// TIA Portal V16 export
// export: Created 2022-11-17T15:49:44.8072382Z, ExportSetting WithDefaults, DisplayName Totally Integrated Automation Portal, DisplayVersion V16 Update 6, DisplayName TIA Portal Version Control Interface, DisplayVersion V16 Update 2, DisplayName TIA Portal Openness, DisplayVersion V16 Update 6, DisplayName SINAMICS Startdrive Advanced, DisplayVersion V16 Update 5, DisplayName SINAMICS Startdrive G130, G150, S120, S150, SINAMICS MV, S210, DisplayVersion V16 Update 5, DisplayName SINAMICS Startdrive G110M, G120, G120C, G120D, G120P, G115D, DisplayVersion V16 Update 5, DisplayName STEP 7 Professional, DisplayVersion V16 Update 6, DisplayName STEP 7 Safety, DisplayVersion V16, DisplayName WinCC Advanced, DisplayVersion V16 Update 6
DATA_BLOCK "DB242_Program8"   // DB242
{ S7_Optimized_Access := 'FALSE' }
AUTHOR : Robopac
VERSION : 0.0
// stored: AutoNumber false, IsOnlyStoredInLoadMemory false, IsWriteProtectedInAS false
   VAR RETAIN
      Program8 { S7_SetPoint := 'True'} : "DatiProgramma";
   END_VAR
BEGIN
   Program8.Wrapping := TRUE;
   Program8.TopLenght := 500;
   Program8.TopRelease := 0;
   Program8.TopDown := 0;
   Program8.Top := 4;
   Program8.PressurePTime := 0;
   Program8.LifterTime := 0;
   Program8.RevOverContrast := 1;
   Program8.RopeEndCycle := 16#02;
   Program8.Spare4 := 16#01;
   Program8.RopeTime := 1500;
   Program8.RevOverClamp := 1;
   Program8.FilmForceFinalRev := 10;
   Program8.FilmPrestretchFinalRev := 100;
   Program8.ArmSpeed := 100;
   Program8.CarriageDown4Top := 500;
   Program8.TopDownTime := 1500;
   Program8.LapsUnderTop := 0;
   Program8.Spare6 := 0;
   Program8.Spare7 := 0;
   Program8.Spare8 := 0;
   Program8.Spare9 := 0;
   Program8.Spare10 := 0;
   Program8.Spare11 := 0;
   Program8.Spare12 := 0;
   Program8.Overlap0_1 := 0;
   Program8.Height1 := 130;
   Program8.Landmark1 := FALSE;
   Program8.Lifter1 := FALSE;
   Program8.SpareBit1H1 := FALSE;
   Program8.Airblower1 := TRUE;
   Program8.NextStep1 := TRUE;
   Program8.PressureP1 := TRUE;
   Program8.SpareByte2H1 := 16#00;
   Program8.Revolution1 := 1;
   Program8.RopeUnit1_1 := 16#01;
   Program8.RopeUnit1_2 := 16#01;
   Program8.FilmForce1 := 5;
   Program8.FilmPrestretch1 := 200;
   Program8.Spare3H1 := 0;
   Program8.Spare49 := 0;
   Program8.Spare50 := 0;
   Program8.Spare51 := 0;
   Program8.Spare52 := 0;
   Program8.Spare53 := 0;
   Program8.Overlap1_2 := 0;
   Program8.Height2 := 50;
   Program8.Landmark2 := FALSE;
   Program8.Lifter2 := FALSE;
   Program8.SpareBit1H2 := FALSE;
   Program8.Airblower2 := TRUE;
   Program8.NextStep2 := TRUE;
   Program8.PressureP2 := TRUE;
   Program8.SpareByte2H2 := 16#00;
   Program8.Revolution2 := 1;
   Program8.RopeUnit2_1 := 16#01;
   Program8.RopeUnit2_2 := 16#01;
   Program8.FilmForce2 := 20;
   Program8.FilmPrestretch2 := 200;
   Program8.Spare3H2 := 0;
   Program8.Spare54 := 0;
   Program8.Spare55 := 0;
   Program8.Spare56 := 0;
   Program8.Spare57 := 0;
   Program8.Spare58 := 0;
   Program8.Overlap2_3 := 100;
   Program8.Height3 := -50;
   Program8.Landmark3 := TRUE;
   Program8.Lifter3 := FALSE;
   Program8.SpareBit1H3 := FALSE;
   Program8.Airblower3 := TRUE;
   Program8.NextStep3 := TRUE;
   Program8.PressureP3 := TRUE;
   Program8.SpareByte2H3 := 16#00;
   Program8.Revolution3 := 2;
   Program8.RopeUnit3_1 := 16#01;
   Program8.RopeUnit3_2 := 16#01;
   Program8.FilmForce3 := 30;
   Program8.FilmPrestretch3 := 200;
   Program8.Spare3H3 := 0;
   Program8.Spare59 := 0;
   Program8.Spare60 := 0;
   Program8.Spare61 := 380;
   Program8.Spare62 := 2800;
   Program8.Spare63 := 0;
   Program8.Overlap3_4 := 100;
   Program8.Height4 := 100;
   Program8.Landmark4 := FALSE;
   Program8.Lifter4 := FALSE;
   Program8.SpareBit1H4 := FALSE;
   Program8.Airblower4 := TRUE;
   Program8.NextStep4 := TRUE;
   Program8.PressureP4 := TRUE;
   Program8.SpareByte2H4 := 16#00;
   Program8.Revolution4 := 3;
   Program8.RopeUnit4_1 := 16#02;
   Program8.RopeUnit4_2 := 16#02;
   Program8.FilmForce4 := 30;
   Program8.FilmPrestretch4 := 200;
   Program8.Spare3H4 := 0;
   Program8.Spare64 := 0;
   Program8.Spare65 := 0;
   Program8.Spare66 := 0;
   Program8.Spare67 := 0;
   Program8.Spare68 := 0;
   Program8.Overlap4_5 := 0;
   Program8.Height5 := 50;
   Program8.Landmark5 := FALSE;
   Program8.Lifter5 := FALSE;
   Program8.SpareBit1H5 := FALSE;
   Program8.Airblower5 := TRUE;
   Program8.NextStep5 := FALSE;
   Program8.PressureP5 := FALSE;
   Program8.SpareByte2H5 := 16#00;
   Program8.Revolution5 := 1;
   Program8.RopeUnit5_1 := 16#01;
   Program8.RopeUnit5_2 := 16#01;
   Program8.FilmForce5 := 30;
   Program8.FilmPrestretch5 := 200;
   Program8.Spare3H5 := 0;
   Program8.Spare69 := 0;
   Program8.Spare70 := 0;
   Program8.Spare71 := 0;
   Program8.Spare72 := 0;
   Program8.Spare73 := 0;
   Program8.Overlap5_6 := 100;
   Program8.Height6 := 50;
   Program8.Landmark6 := FALSE;
   Program8.Lifter6 := FALSE;
   Program8.SpareBit1H6 := FALSE;
   Program8.Airblower6 := TRUE;
   Program8.NextStep6 := FALSE;
   Program8.PressureP6 := FALSE;
   Program8.SpareByte2H6 := 16#00;
   Program8.Revolution6 := 2;
   Program8.RopeUnit6_1 := 16#02;
   Program8.RopeUnit6_2 := 16#01;
   Program8.FilmForce6 := 20;
   Program8.FilmPrestretch6 := 200;
   Program8.Spare3H6 := 0;
   Program8.Spare74 := 0;
   Program8.Spare75 := 0;
   Program8.Spare76 := 0;
   Program8.Spare77 := 0;
   Program8.Spare78 := 0;
   Program8.Overlap6_7 := 0;
   Program8.Height7 := 0;
   Program8.Landmark7 := FALSE;
   Program8.Lifter7 := FALSE;
   Program8.SpareBit1H7 := FALSE;
   Program8.Airblower7 := FALSE;
   Program8.NextStep7 := TRUE;
   Program8.PressureP7 := FALSE;
   Program8.SpareByte2H7 := 16#00;
   Program8.Revolution7 := 1;
   Program8.RopeUnit7_1 := 16#01;
   Program8.RopeUnit7_2 := 16#01;
   Program8.FilmForce7 := 0;
   Program8.FilmPrestretch7 := 100;
   Program8.Spare3H7 := 0;
   Program8.Spare79 := 0;
   Program8.Spare80 := 0;
   Program8.Spare81 := 0;
   Program8.Spare82 := 0;
   Program8.Spare83 := 0;
   Program8.Overlap7_8 := 0;
   Program8.Height8 := 0;
   Program8.Landmark8 := FALSE;
   Program8.Lifter8 := FALSE;
   Program8.SpareBit1H8 := FALSE;
   Program8.Airblower8 := FALSE;
   Program8.NextStep8 := TRUE;
   Program8.PressureP8 := FALSE;
   Program8.SpareByte2H8 := 16#00;
   Program8.Revolution8 := 1;
   Program8.RopeUnit8_1 := 16#01;
   Program8.RopeUnit8_2 := 16#01;
   Program8.FilmForce8 := 0;
   Program8.FilmPrestretch8 := 100;
   Program8.Spare3H8 := 0;
   Program8.Spare84 := 0;
   Program8.Spare85 := 0;
   Program8.Spare86 := 0;
   Program8.Spare87 := 0;
   Program8.Spare88 := 0;
   Program8.Overlap8_9 := 0;
   Program8.Height9 := 0;
   Program8.Landmark9 := FALSE;
   Program8.Lifter9 := FALSE;
   Program8.SpareBit1H9 := FALSE;
   Program8.Airblower9 := FALSE;
   Program8.NextStep9 := TRUE;
   Program8.PressureP9 := FALSE;
   Program8.SpareByte2H9 := 16#00;
   Program8.Revolution9 := 1;
   Program8.RopeUnit9_1 := 16#01;
   Program8.RopeUnit9_2 := 16#01;
   Program8.FilmForce9 := 0;
   Program8.FilmPrestretch9 := 100;
   Program8.Spare3H9 := 0;
   Program8.Spare89 := 0;
   Program8.Spare90 := 0;
   Program8.Spare91 := 0;
   Program8.Spare92 := 0;
   Program8.Spare93 := 0;
   Program8.Overlap9_10 := 0;
   Program8.Height10 := 0;
   Program8.Landmark10 := FALSE;
   Program8.Lifter10 := FALSE;
   Program8.SpareBit1H10 := FALSE;
   Program8.Airblower10 := FALSE;
   Program8.NextStep10 := FALSE;
   Program8.PressureP10 := FALSE;
   Program8.SpareByte2H10 := 16#00;
   Program8.Revolution10 := 1;
   Program8.RopeUnit10_1 := 16#01;
   Program8.RopeUnit10_2 := 16#01;
   Program8.FilmForce10 := 0;
   Program8.FilmPrestretch10 := 100;
   Program8.Spare3H10 := 0;
   Program8.Spare94 := 0;
   Program8.Spare95 := 0;
   Program8.Spare96 := 0;
   Program8.Spare97 := 0;
   Program8.Spare98 := 0;
   Program8.Overlap10_11 := 0;
   Program8.Height11 := 0;
   Program8.Landmark11 := FALSE;
   Program8.Lifter11 := FALSE;
   Program8.SpareBit1H11 := FALSE;
   Program8.Airblower11 := FALSE;
   Program8.NextStep11 := TRUE;
   Program8.PressureP11 := FALSE;
   Program8.SpareByte2H11 := 16#00;
   Program8.Revolution11 := 1;
   Program8.RopeUnit11_1 := 16#01;
   Program8.RopeUnit11_2 := 16#01;
   Program8.FilmForce11 := 0;
   Program8.FilmPrestretch11 := 100;
   Program8.Spare3H11 := 0;
   Program8.Spare99 := 0;
   Program8.Spare100 := 0;
   Program8.Spare101 := 0;
   Program8.Spare102 := 0;
   Program8.Spare103 := 0;
   Program8.Overlap11_12 := 0;
   Program8.Height12 := 0;
   Program8.Landmark12 := FALSE;
   Program8.Lifter12 := FALSE;
   Program8.SpareBit1H12 := FALSE;
   Program8.Airblower12 := FALSE;
   Program8.NextStep12 := FALSE;
   Program8.PressureP12 := FALSE;
   Program8.SpareByte2H12 := 16#00;
   Program8.Revolution12 := 1;
   Program8.RopeUnit12_1 := 16#01;
   Program8.RopeUnit12_2 := 16#01;
   Program8.FilmForce12 := 0;
   Program8.FilmPrestretch12 := 100;
   Program8.Spare3H12 := 0;
   Program8.Spare104 := 0;
   Program8.Spare105 := 0;
   Program8.Spare106 := 0;
   Program8.Spare107 := 0;
   Program8.Spare108 := 0;
END_DATA_BLOCK
